# EPICS alarm handler configuration: mps_database/bareTest/alarms/areas/mpln_l0b_mp05.alhConfig
GROUP NULL MPLN:L0B:MP05:1
$ALIAS MPS Link Node 55
$GUIDANCE
LTUH MPS
   Group Name: MPLN:L0B:MP05:1
   Summary PV:  MPLN:L0B:MP05:1:STATSUMY
$END
CHANNEL  MPLN:L0B:MP05:1    MPLN:L0B:MP05:1:MPS_EN_RBV		-----
CHANNEL  MPLN:L0B:MP05:1    MPLN:L0B:MP05:1:LC1_MODE_RBV		-----
